// TIA Portal project "Traffic Lights" (V17)

(* hardware
DEVICE "S7-1500/ET200MP station_1"  S7-1500 station
   slot 0: "Rail_0"  Rack  6ES7 590-1***0-0AA0
   slot 1: "PLC_1"  CPU 1512C-1 PN  6ES7 512-1CK01-0AB0  V2.9
      slot 3: "CPU display_1"  6ES7591-1AA00-0AA0
      slot 32768: "PROFINET interface_1"  X1
         slot 32769: "Port_1"  X1 P1
         slot 32770: "Port_2"  X1 P2
      slot 34817: "Virtual CP interface port_1"  Virtual CP interface port  Virtual CP interface port
*)

// ===== PLC "PLC_1"  CPU 1512C-1 PN =====

VAR_GLOBAL   // PLC tag table "Default tag table"
   "StartSystem" AT %M0.0 : Bool;
   "SET" AT %M0.1 : Bool;
END_VAR

TYPE "Traffic_Lights"
   STRUCT
      Red_Light : Bool;
      Yellow_Light : Bool;
      Green_Light : Bool;
   END_STRUCT;
END_TYPE

DATA_BLOCK "Traffic_Lights_DB"   // DB1
{ S7_Optimized_Access := 'TRUE' }
VERSION : 0.1
   VAR
      Northern_TrafficLights : "Traffic_Lights";
      Southern_TrafficLights : "Traffic_Lights";
      Eastern_TrafficLights : "Traffic_Lights";
      Western_TrafficLights : "Traffic_Lights";
      Start : Bool;
      Stop : Bool;
   END_VAR
BEGIN
END_DATA_BLOCK

// folder: System blocks/Program resources

DATA_BLOCK "IEC_Timer_0_DB"   // DB2
{ S7_Optimized_Access := 'TRUE' }
AUTHOR : Simatic
FAMILY : IEC
NAME : IEC_TMR
VERSION : 1.0
// stored: InstanceOfName IEC_TIMER
"IEC_TIMER"
BEGIN
END_DATA_BLOCK

DATA_BLOCK "IEC_Timer_0_DB_2"   // DB4
{ S7_Optimized_Access := 'TRUE' }
AUTHOR : Simatic
FAMILY : IEC
NAME : IEC_TMR
VERSION : 1.0
// stored: InstanceOfName IEC_TIMER
"IEC_TIMER"
BEGIN
END_DATA_BLOCK

DATA_BLOCK "IEC_Timer_0_DB_3"   // DB5
{ S7_Optimized_Access := 'TRUE' }
AUTHOR : Simatic
FAMILY : IEC
NAME : IEC_TMR
VERSION : 1.0
// stored: InstanceOfName IEC_TIMER
"IEC_TIMER"
BEGIN
END_DATA_BLOCK

DATA_BLOCK "IEC_Timer_0_DB_4"   // DB6
{ S7_Optimized_Access := 'TRUE' }
AUTHOR : Simatic
FAMILY : IEC
NAME : IEC_TMR
VERSION : 1.0
// stored: InstanceOfName IEC_TIMER
"IEC_TIMER"
BEGIN
END_DATA_BLOCK

// folder: (top level)

FUNCTION "Traffic_Lights_FC" : Void   // FC1, LAD
{ S7_Optimized_Access := 'TRUE' }
VERSION : 0.1
   VAR_INPUT
      Start_PB : Bool;
      Stop_PB : Bool;
   END_VAR
   VAR_OUTPUT
      "Red_Light_North/South" : Bool;
      "Green_Light_North/South" : Bool;
      "Red_Light_East/West" : Bool;
      "Green_Light_East/West" : Bool;
      "Yellow_Light_North/South" : Bool;
      "Yellow_Light_East/West" : Bool;
   END_VAR
BEGIN

REGION Network 1: START TRAFFIC LIGHTS
   // This Block Starts and Stops the whole trafficl lights system. The SR block acts as a latch for the momentary start push buttons
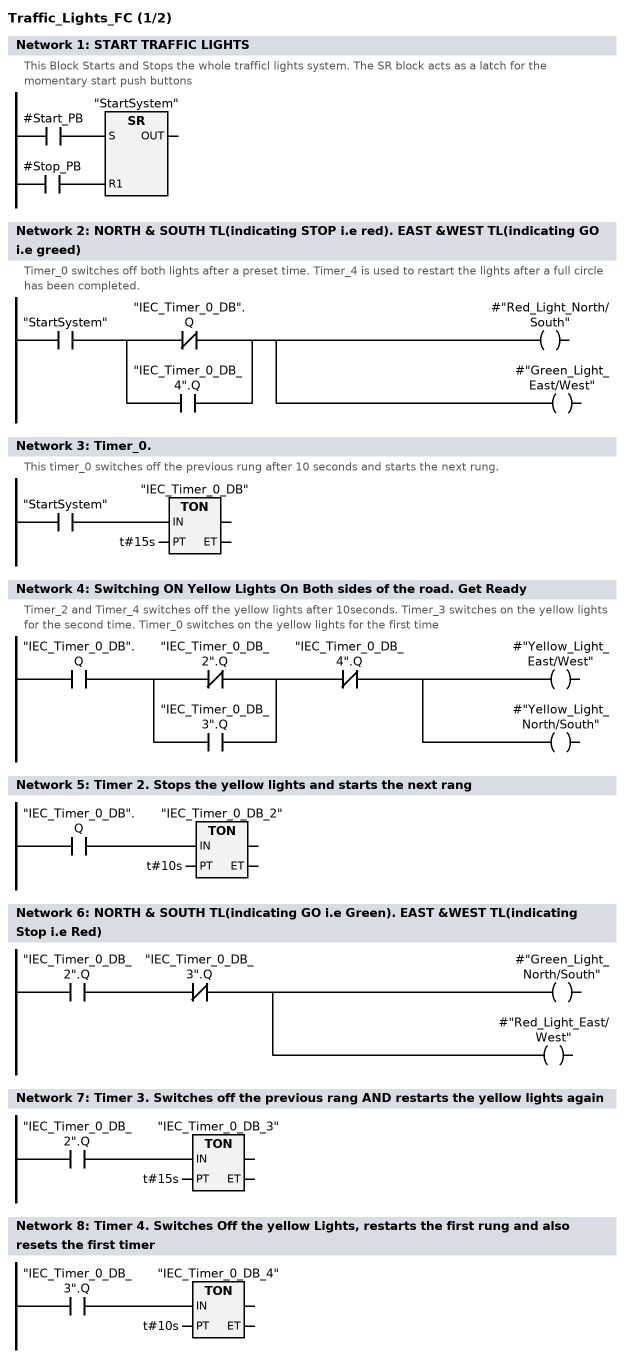
   RUNG wire#powerrail
      Contact( #Start_PB )
      S_SR(operand := "StartSystem", r1 := wire#w1)
   END_RUNG
   RUNG wire#powerrail
      Contact( #Stop_PB )
   END_RUNG wire#w1
   // the same network as SCL:
   IF #Start_PB THEN
       "StartSystem" := TRUE;   // SR flip-flop
   END_IF;
   IF #Stop_PB THEN "StartSystem" := FALSE; END_IF;
END_REGION

REGION Network 2: NORTH & SOUTH TL(indicating STOP i.e red). EAST &WEST TL(indicating GO i.e greed)
   // Timer_0 switches off both lights after a preset time. Timer_4 is used to restart the lights after a full circle has been completed.
   RUNG wire#powerrail
      Contact( "StartSystem" )
      wire#w1
      I_Contact( "IEC_Timer_0_DB".Q )
      wire#w2
      Coil( #"Red_Light_North/South" )
   END_RUNG
   RUNG wire#w1
      Contact( "IEC_Timer_0_DB_4".Q )
   END_RUNG wire#w2
   RUNG wire#w2
      Coil( #"Green_Light_East/West" )
   END_RUNG
   // the same network as SCL:
   #"Red_Light_North/South" := "StartSystem" AND (NOT "IEC_Timer_0_DB".Q OR "IEC_Timer_0_DB_4".Q);
   #"Green_Light_East/West" := #"Red_Light_North/South";
END_REGION

REGION Network 3: Timer_0.
   // This timer_0 switches off the previous rung after 10 seconds and starts the next rung.
   "IEC_Timer_0_DB".TON(IN := "StartSystem", PT := t#15s);
END_REGION

REGION Network 4: Switching ON Yellow Lights On Both sides of the road. Get Ready
   // Timer_2 and Timer_4 switches off the yellow lights after 10seconds. Timer_3 switches on the yellow lights for the second time. Timer_0 switches on the yellow lights for the first time
   RUNG wire#powerrail
      Contact( "IEC_Timer_0_DB".Q )
      wire#w1
      I_Contact( "IEC_Timer_0_DB_2".Q )
      wire#w2
      I_Contact( "IEC_Timer_0_DB_4".Q )
      wire#w3
      Coil( #"Yellow_Light_East/West" )
   END_RUNG
   RUNG wire#w1
      Contact( "IEC_Timer_0_DB_3".Q )
   END_RUNG wire#w2
   RUNG wire#w3
      Coil( #"Yellow_Light_North/South" )
   END_RUNG
   // the same network as SCL:
   #"Yellow_Light_East/West" := "IEC_Timer_0_DB".Q AND (NOT "IEC_Timer_0_DB_2".Q OR "IEC_Timer_0_DB_3".Q) AND NOT "IEC_Timer_0_DB_4".Q;
   #"Yellow_Light_North/South" := #"Yellow_Light_East/West";
END_REGION

REGION Network 5: Timer 2. Stops the yellow lights and starts the next rang
   "IEC_Timer_0_DB_2".TON(IN := "IEC_Timer_0_DB".Q, PT := t#10s);
END_REGION

REGION Network 6: NORTH & SOUTH TL(indicating GO i.e Green). EAST &WEST TL(indicating Stop i.e Red)
   RUNG wire#powerrail
      Contact( "IEC_Timer_0_DB_2".Q )
      I_Contact( "IEC_Timer_0_DB_3".Q )
      wire#w1
      Coil( #"Green_Light_North/South" )
   END_RUNG
   RUNG wire#w1
      Coil( #"Red_Light_East/West" )
   END_RUNG
   // the same network as SCL:
   #"Green_Light_North/South" := "IEC_Timer_0_DB_2".Q AND NOT "IEC_Timer_0_DB_3".Q;
   #"Red_Light_East/West" := #"Green_Light_North/South";
END_REGION

REGION Network 7: Timer 3. Switches off the previous rang AND restarts the yellow lights again
   "IEC_Timer_0_DB_3".TON(IN := "IEC_Timer_0_DB_2".Q, PT := t#15s);
END_REGION

REGION Network 8: Timer 4. Switches Off the yellow Lights, restarts the first rung and also resets the first timer
   "IEC_Timer_0_DB_4".TON(IN := "IEC_Timer_0_DB_3".Q, PT := t#10s);
END_REGION

REGION Network 9: Reseting the first timer to allow new time count
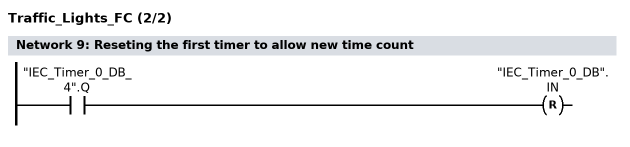
   RUNG wire#powerrail
      Contact( "IEC_Timer_0_DB_4".Q )
      R_Coil( "IEC_Timer_0_DB".IN )
   END_RUNG
   // the same network as SCL:
   IF "IEC_Timer_0_DB_4".Q THEN "IEC_Timer_0_DB".IN := FALSE; END_IF;
END_REGION
END_FUNCTION

ORGANIZATION_BLOCK "Main"   // OB1, LAD, ProgramCycle
TITLE = "Main Program Sweep (Cycle)"
{ S7_Optimized_Access := 'TRUE' }
VERSION : 0.1
   VAR_INPUT
      Initial_Call : Bool;   // Initial call of this OB
      Remanence : Bool;   // =True, if remanent data are available
   END_VAR
BEGIN

REGION Network 1: Northern Side And Eastern Side Block
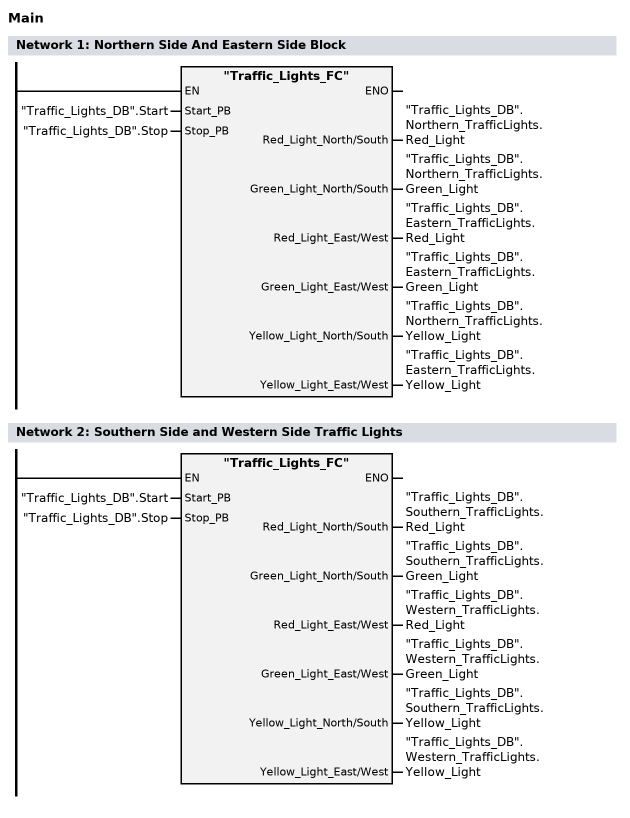
   RUNG wire#powerrail
      "Traffic_Lights_FC"(Start_PB := "Traffic_Lights_DB".Start, Stop_PB := "Traffic_Lights_DB".Stop, "Red_Light_North/South" => "Traffic_Lights_DB".Northern_TrafficLights.Red_Light, "Green_Light_North/South" => "Traffic_Lights_DB".Northern_TrafficLights.Green_Light, "Red_Light_East/West" => "Traffic_Lights_DB".Eastern_TrafficLights.Red_Light, "Green_Light_East/West" => "Traffic_Lights_DB".Eastern_TrafficLights.Green_Light, "Yellow_Light_North/South" => "Traffic_Lights_DB".Northern_TrafficLights.Yellow_Light, "Yellow_Light_East/West" => "Traffic_Lights_DB".Eastern_TrafficLights.Yellow_Light)
   END_RUNG
   // the same network as SCL:
   "Traffic_Lights_FC"(Start_PB := "Traffic_Lights_DB".Start,
                       Stop_PB := "Traffic_Lights_DB".Stop,
                       "Red_Light_North/South" => "Traffic_Lights_DB".Northern_TrafficLights.Red_Light,
                       "Green_Light_North/South" => "Traffic_Lights_DB".Northern_TrafficLights.Green_Light,
                       "Red_Light_East/West" => "Traffic_Lights_DB".Eastern_TrafficLights.Red_Light,
                       "Green_Light_East/West" => "Traffic_Lights_DB".Eastern_TrafficLights.Green_Light,
                       "Yellow_Light_North/South" => "Traffic_Lights_DB".Northern_TrafficLights.Yellow_Light,
                       "Yellow_Light_East/West" => "Traffic_Lights_DB".Eastern_TrafficLights.Yellow_Light);
END_REGION

REGION Network 2: Southern Side and Western Side Traffic Lights
   RUNG wire#powerrail
      "Traffic_Lights_FC"(Start_PB := "Traffic_Lights_DB".Start, Stop_PB := "Traffic_Lights_DB".Stop, "Red_Light_North/South" => "Traffic_Lights_DB".Southern_TrafficLights.Red_Light, "Green_Light_North/South" => "Traffic_Lights_DB".Southern_TrafficLights.Green_Light, "Red_Light_East/West" => "Traffic_Lights_DB".Western_TrafficLights.Red_Light, "Green_Light_East/West" => "Traffic_Lights_DB".Western_TrafficLights.Green_Light, "Yellow_Light_North/South" => "Traffic_Lights_DB".Southern_TrafficLights.Yellow_Light, "Yellow_Light_East/West" => "Traffic_Lights_DB".Western_TrafficLights.Yellow_Light)
   END_RUNG
   // the same network as SCL:
   "Traffic_Lights_FC"(Start_PB := "Traffic_Lights_DB".Start,
                       Stop_PB := "Traffic_Lights_DB".Stop,
                       "Red_Light_North/South" => "Traffic_Lights_DB".Southern_TrafficLights.Red_Light,
                       "Green_Light_North/South" => "Traffic_Lights_DB".Southern_TrafficLights.Green_Light,
                       "Red_Light_East/West" => "Traffic_Lights_DB".Western_TrafficLights.Red_Light,
                       "Green_Light_East/West" => "Traffic_Lights_DB".Western_TrafficLights.Green_Light,
                       "Yellow_Light_North/South" => "Traffic_Lights_DB".Southern_TrafficLights.Yellow_Light,
                       "Yellow_Light_East/West" => "Traffic_Lights_DB".Western_TrafficLights.Yellow_Light);
END_REGION
END_ORGANIZATION_BLOCK